FUNCTION_BLOCK TemplateBasicEmpty (* Basic FB with empty ECC *)
  (* Standard: 61499-2 *)
  (* Version 1.0, 2016-05-26, AZ, fortiss GmbH *)
  EC_STATES
    START; (* Initial State *)
  END_STATES
END_FUNCTION_BLOCK
